TYPE AxesTabs :
(
	OVERVIEW := 0,
	MANUAL := 1,
    AXES := 2,
	TARGET := 3,
    TPOINT := 4,
    ADVANCED := 5,
    IO := 6,
    CONFIG := 7
);
END_TYPE

(* stored: Version 1.1.0.1, ProductVersion 3.1.4018.5
   DUT AxesTabs: Id {20e939ad-5749-44d1-94ff-32045bbbef99} *)
